{attribute addProperty BoxType "EK1100-0000-0018"}
{attribute addProperty Id "Beckhoff_ELM36xxEK1122Beckhoff_ELM36xxEK1122_DABD45E4162A_0001_ELM3602_0000_0017ELM3602_08F8D9E433842.25A_0002_ELM3602_0000_0018ELM3602_08F8D9E433842.25A_0003_ELM3602_0002_0016ELM3602_08F8D9E433842.25A_0004_ELM3602_0002_0017ELM3602_08F8D9E433842.25A_0005_ELM3602_0002_0018ELM3602_08F8D9E433842.25A_0006_ELM3604_0000_0017ELM3604_B740F21646658.25A_0007_ELM3604_0000_0018ELM3604_B740F21646658.25A_0008_ELM3604_0002_0016ELM3604_B740F21646658.25A_0009_ELM3604_0002_0017ELM3604_B740F21646658.25A_0010_ELM3604_0002_0018ELM3604_B740F21646658.25"}
{attribute addProperty CRC "4110695804"}
{attribute addProperty SizeInBites "4036"}
{attribute addProperty SizeInBytes "504.5"}
TYPE Beckhoff_ELM36xx_F5043D7C EXTENDS EK1100_179A0949 :
STRUCT
	{attribute addProperty Name "Beckhoff_ELM36xxEK1122"}
	Beckhoff_ELM36xxEK1122 : Beckhoff_ELM36xxEK1122_DABD45E4;
	{attribute addProperty Name "A_0001_ELM3602_0000_0017"}
	A_0001_ELM3602_0000_0017 : ELM3602_08F8D9E4;
	{attribute addProperty Name "A_0002_ELM3602_0000_0018"}
	A_0002_ELM3602_0000_0018 : ELM3602_08F8D9E4;
	{attribute addProperty Name "A_0003_ELM3602_0002_0016"}
	A_0003_ELM3602_0002_0016 : ELM3602_08F8D9E4;
	{attribute addProperty Name "A_0004_ELM3602_0002_0017"}
	A_0004_ELM3602_0002_0017 : ELM3602_08F8D9E4;
	{attribute addProperty Name "A_0005_ELM3602_0002_0018"}
	A_0005_ELM3602_0002_0018 : ELM3602_08F8D9E4;
	{attribute addProperty Name "A_0006_ELM3604_0000_0017"}
	A_0006_ELM3604_0000_0017 : ELM3604_B740F216;
	{attribute addProperty Name "A_0007_ELM3604_0000_0018"}
	A_0007_ELM3604_0000_0018 : ELM3604_B740F216;
	{attribute addProperty Name "A_0008_ELM3604_0002_0016"}
	A_0008_ELM3604_0002_0016 : ELM3604_B740F216;
	{attribute addProperty Name "A_0009_ELM3604_0002_0017"}
	A_0009_ELM3604_0002_0017 : ELM3604_B740F216;
	{attribute addProperty Name "A_0010_ELM3604_0002_0018"}
	A_0010_ELM3604_0002_0018 : ELM3604_B740F216;
END_STRUCT
END_TYPE

(* stored: Version 1.2.0.0, ProductVersion 3.1.4024.9
   DUT Beckhoff_ELM36xx_F5043D7C: Id {072969ee-d925-49df-a03e-1f3ca2ae998f} *)
